TYPE Vec5b : ARRAY[1..5] OF bool; END_TYPE

(* stored: Version 1.1.0.1, ProductVersion 3.1.4024.12
   DUT Vec5b: Id {240fa815-2303-488d-a2e9-17abbcd31a03} *)
